FUNCTION_BLOCK ST_CREATE_CONN (* Creates an event or data connection between two FB instances *)
  (* Standard: 61499-1; Classification: Reconfiguration; Function: Creates Connection; Type: Structural Service; Description: Copyright (c) 2012 Profactor GmbH This program and the accompanying materials are made available under the terms of the Eclipse Public License 2.0 which is available at https://www.eclipse.org/legal/epl-2.0/ SPDX-License-Identifier: EPL-2.0 *)
  (* Version 3.0, 2025-04-14, Patrick Aigner, changed package *)
  (* Version 1.0, 2012-05-31, Gerhard Ebenhofer, Profactor GmbH *)
  PACKAGE eclipse4diac::reconfiguration;
  (* Compiler Cpp GNU GCC >3.0 *)
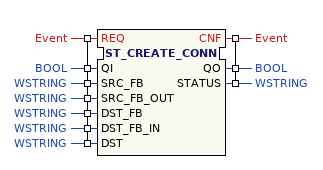
  EVENT_INPUT
    REQ WITH SRC_FB, SRC_FB_OUT, DST_FB, DST_FB_IN, DST, QI; (* Event to require creation of a connection *)
  END_EVENT
  EVENT_OUTPUT
    CNF WITH STATUS, QO; (* Event to confirm that the connection has been created *)
  END_EVENT
  VAR_INPUT
    QI : BOOL; (* Event Input Qualifier *)
    SRC_FB : WSTRING; (* Reference to Source FB instance *)
    SRC_FB_OUT : WSTRING; (* Reference to Source FB instance Event/Data-Output *)
    DST_FB : WSTRING; (* Reference to Destination FB instance *)
    DST_FB_IN : WSTRING; (* Reference to Destination FB instance Event/Data-Input *)
    DST : WSTRING; (* Destination where the connection has to be created (Syntax: ResourceName) *)
  END_VAR
  VAR_OUTPUT
    QO : BOOL; (* Event Output Qualifier *)
    STATUS : WSTRING; (* Service Status: RDY, NO_SUCH_OBJECT, INVALID_STATE *)
  END_VAR
  SERVICE APPLICATION/RESOURCE
    SEQUENCE normal_establishment
      APPLICATION.INIT+() -> APPLICATION.INITO+();
    END_SEQUENCE
    SEQUENCE unsuccessful_establishment
      APPLICATION.INIT+() -> APPLICATION.INITO-();
    END_SEQUENCE
    SEQUENCE request_confirm
      APPLICATION.REQ+() -> APPLICATION.CNF+();
    END_SEQUENCE
    SEQUENCE request_inhibited
      APPLICATION.REQ-() -> APPLICATION.CNF-();
    END_SEQUENCE
    SEQUENCE request_error
      APPLICATION.REQ+() -> APPLICATION.CNF-();
    END_SEQUENCE
    SEQUENCE application_initiated_termination
      APPLICATION.INIT-() -> APPLICATION.INITO-();
    END_SEQUENCE
    SEQUENCE resource_initiated_termination
      -> APPLICATION.INITO-();
    END_SEQUENCE
  END_SERVICE
END_FUNCTION_BLOCK
